FUNCTION F_RoundLrealEx : LREAL
VAR_INPUT
	lrIn : LREAL;
	iPrecision : UINT;
END_VAR
VAR
	lrTemp	: LREAL;
END_VAR

lrTemp := lrIn * EXPT(10,iPrecision);
lrTemp := LTRUNC(lrTemp);
F_RoundLrealEx := lrTemp / EXPT(10,iPrecision);

END_FUNCTION

(* stored: Version 1.1.0.1, ProductVersion 3.1.4024.12
   POU F_RoundLrealEx: Id {0587239f-475c-4921-beb6-3f0e2e60f459}, SpecialFunc None *)
